// Mitsubishi GX Works2 project: 시퀀스 회로 예제 (타이머, 카운터)   PLC: Q03UDV

PROGRAM MAIN
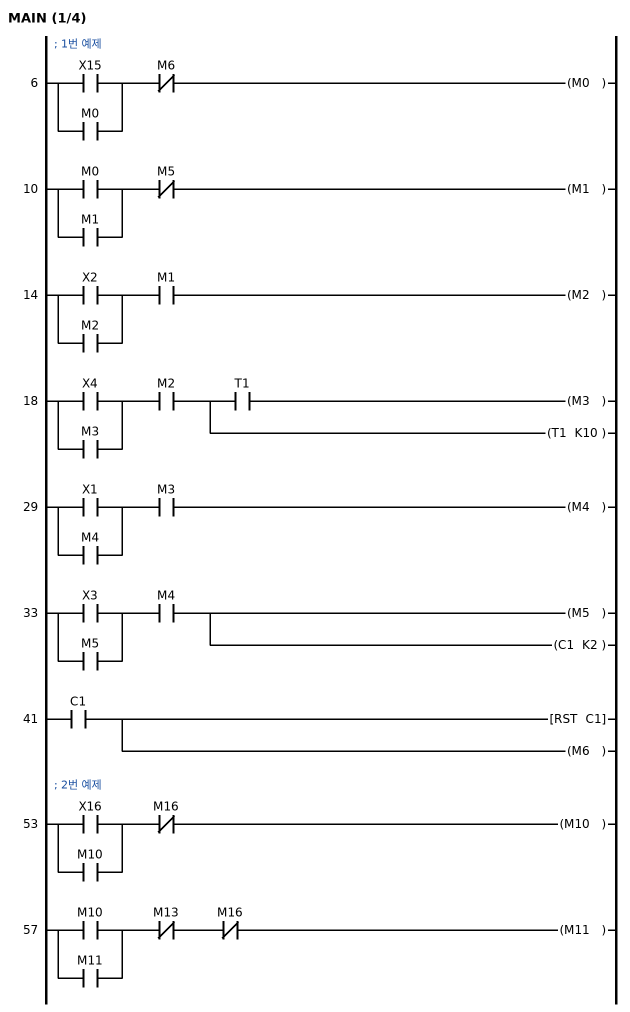
; 1번 예제
6     LD      X15
      OR      M0
      ANI     M6
      OUT     M0
10    LD      M0
      OR      M1
      ANI     M5
      OUT     M1
14    LD      X2
      OR      M2
      AND     M1
      OUT     M2
18    LD      X4
      OR      M3
      AND     M2
      MPS
      AND     T1
      OUT     M3
      MPP
      OUT     T1 K10
29    LD      X1
      OR      M4
      AND     M3
      OUT     M4
33    LD      X3
      OR      M5
      AND     M4
      OUT     M5
      OUT     C1 K2
41    LD      C1
      RST     C1
      OUT     M6
; 2번 예제
53    LD      X16
      OR      M10
      ANI     M16
      OUT     M10
57    LD      M10
      OR      M11
      ANI     M13
      ANI     M16
      OUT     M11
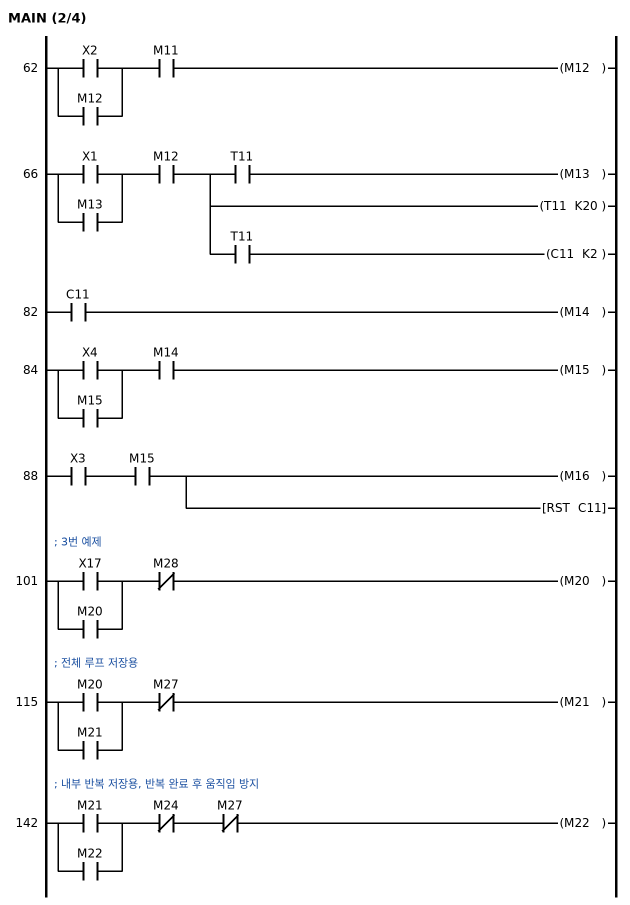
62    LD      X2
      OR      M12
      AND     M11
      OUT     M12
66    LD      X1
      OR      M13
      AND     M12
      MPS
      AND     T11
      OUT     M13
      MPP
      OUT     T11 K20
      AND     T11
      OUT     C11 K2
82    LD      C11
      OUT     M14
84    LD      X4
      OR      M15
      AND     M14
      OUT     M15
88    LD      X3
      AND     M15
      OUT     M16
      RST     C11
; 3번 예제
101   LD      X17
      OR      M20
      ANI     M28
      OUT     M20
; 전체 루프 저장용
115   LD      M20
      OR      M21
      ANI     M27
      OUT     M21
; 내부 반복 저장용, 반복 완료 후 움직임 방지
142   LD      M21
      OR      M22
      ANI     M24
      ANI     M27
      OUT     M22
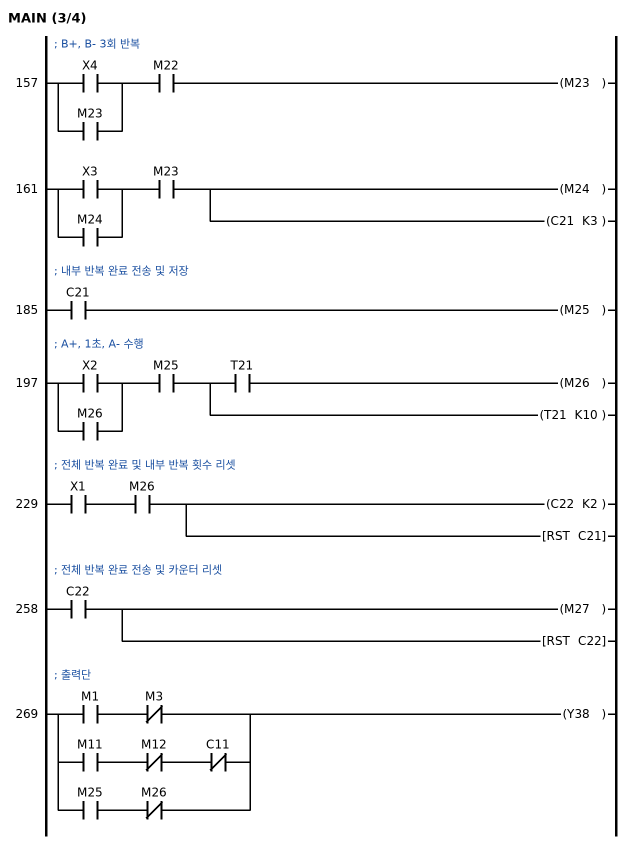
; B+, B- 3회 반복
157   LD      X4
      OR      M23
      AND     M22
      OUT     M23
161   LD      X3
      OR      M24
      AND     M23
      OUT     M24
      OUT     C21 K3
; 내부 반복 완료 전송 및 저장
185   LD      C21
      OUT     M25
; A+, 1초, A- 수행
197   LD      X2
      OR      M26
      AND     M25
      MPS
      AND     T21
      OUT     M26
      MPP
      OUT     T21 K10
; 전체 반복 완료 및 내부 반복 횟수 리셋
229   LD      X1
      AND     M26
      OUT     C22 K2
      RST     C21
; 전체 반복 완료 전송 및 카운터 리셋
258   LD      C22
      OUT     M27
      RST     C22
; 출력단
269   LD      M1
      ANI     M3
      LD      M11
      ANI     M12
      ANI     C11
      ORB
      LD      M25
      ANI     M26
      ORB
      OUT     Y38
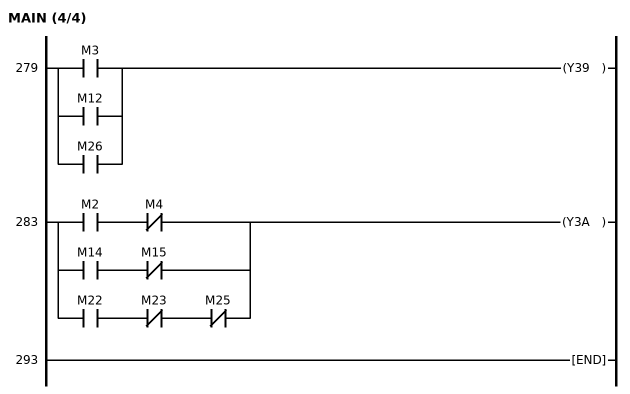
279   LD      M3
      OR      M12
      OR      M26
      OUT     Y39
283   LD      M2
      ANI     M4
      LD      M14
      ANI     M15
      ORB
      LD      M22
      ANI     M23
      ANI     M25
      ORB
      OUT     Y3A
293   END
END_PROGRAM
